// Mitsubishi GX Works2 project: One shot ladder 2   PLC: Q03UDV

PROGRAM MAIN
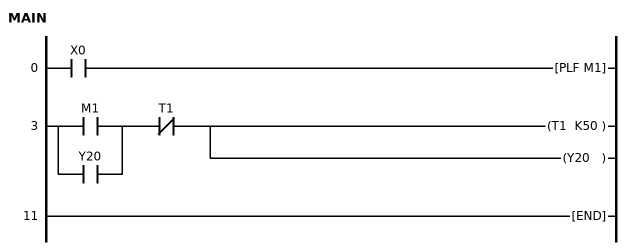
0     LD      X0
      PLF     M1
3     LD      M1
      OR      Y20
      ANI     T1
      OUT     T1 K50
      OUT     Y20
11    END
END_PROGRAM
